{attribute 'qualified_only'}
VAR_GLOBAL
	
	ncAxis1:AXIS_REF; //define axis ref
	plcAxis1:typeDriveInterface; //plc ref inside to be sent to FB_DriveInterface
	
	ncAxis2:AXIS_REF; //define axis ref
	plcAxis2:typeDriveInterface; //plc ref inside to be sent to FB_DriveInterface

	ncAxis3:AXIS_REF; //define axis ref
	plcAxis3:typeDriveInterface; //plc ref inside to be sent to FB_DriveInterface

	ncAxis4:AXIS_REF; //define axis ref
	plcAxis4:typeDriveInterface; //plc ref inside to be sent to FB_DriveInterface
	
	ncAxis5:AXIS_REF; //define axis ref
	plcAxis5:typeDriveInterface; //plc ref inside to be sent to FB_DriveInterface

	ncAxis6:AXIS_REF; //define axis ref
	plcAxis6:typeDriveInterface; //plc ref inside to be sent to FB_DriveInterface

	ncAxis7:AXIS_REF; //define axis ref
	plcAxis7:typeDriveInterface; //plc ref inside to be sent to FB_DriveInterface
	
	ncAxis8:AXIS_REF; //define axis ref
	plcAxis8:typeDriveInterface; //plc ref inside to be sent to FB_DriveInterface

	ncAxis9:AXIS_REF; //define axis ref
	plcAxis9:typeDriveInterface; //plc ref inside to be sent to FB_DriveInterface

	ncAxis10:AXIS_REF; //define axis ref
	plcAxis10:typeDriveInterface; //plc ref inside to be sent to FB_DriveInterface


	//HMI view
	hmiAxis:AXIS_REF; //define axis ref
	
	hmiAxisSel:UINT; //selected index
	tAxisList:ARRAY[1..99] OF STRING(80); //text contents of axis

END_VAR

(* stored: Version 1.1.0.1, ProductVersion 3.1.4024.12
   GVL driveGlobals: Id {1abbc8a1-9bd6-44f7-8544-885342ba4989} *)
